// TIA Portal V17 export
// export: Created 2022-12-08T10:14:51.5933257Z, ExportSetting WithDefaults, DisplayName Totally Integrated Automation Portal, DisplayVersion V17 Update 5, DisplayName TIA Portal Openness, DisplayVersion V17 Update 5, DisplayName TIA Portal Version Control Interface, DisplayVersion V17, DisplayName Simotion SCOUT TIA, DisplayVersion 5.4.3.0, DisplayName SINAMICS Startdrive Advanced, DisplayVersion V17 SP1, DisplayName SINAMICS Startdrive G130, G150, S120, S150, SINAMICS MV, S210, DisplayVersion V17 SP1, DisplayName SINAMICS Startdrive G110M, G120, G120C, G120D, G120P, G115D, DisplayVersion V17 SP1, DisplayName STEP 7 Professional, DisplayVersion V17 Update 5, DisplayName STEP 7 Safety, DisplayVersion V17, DisplayName WinCC Advanced, DisplayVersion V17 Update 5
DATA_BLOCK "DB_Glueing"   // DB20
VERSION : 0.1
// stored: AutoNumber true, DBAccessibleFromOPCUA true, DBAccessibleFromWebserver true, InstanceOfName FB_Glueing, InstanceOfType FB
"FB_Glueing"
   // VAR_INPUT
   //    i_Axis : Array["LOWERAXISNUMBER".."UPPERAXISNUMBER"] of DB_ANY;
   //    i_ActualData : Array["LOWERAXISNUMBER".."UPPERAXISNUMBER"] of "UDT_ServoActualData";
   //    i_Reset : Bool;
   //    i_GlueingEnable : Bool;
   //    i_AxesEnabled : Bool;
   //    i_DetectKarton_1 : Bool;
   //    i_DetectKarton_2 : Bool;
   //    i_DetectKarton_3 : Bool;
   //    i_DetectKarton_4 : Bool;
   //    i_DetectKarton_5 : Bool;
   //    i_DetectKarton_6 : Bool;
   //    i_DetectKarton_7 : Bool;
   //    i_DetectKarton_8 : Bool;
   //    i_MasterAxisForGlueing : Int;
   //    i_MaxNumberOfGlueing : Int;
   // END_VAR
   // VAR_OUTPUT
   //    q_TrackOutput_1 : Bool;
   //    q_TrackOutput_2 : Bool;
   //    q_TrackOutput_3 : Bool;
   //    q_TrackOutput_4 : Bool;
   //    q_TrackOutput_5 : Bool;
   //    q_TrackOutput_6 : Bool;
   //    q_TrackOutput_7 : Bool;
   //    q_TrackOutput_8 : Bool;
   //    q_SensorPermanentlyOccupied_1 : Bool;
   //    q_SensorPermanentlyOccupied_2 : Bool;
   //    q_SensorPermanentlyOccupied_3 : Bool;
   //    q_SensorPermanentlyOccupied_4 : Bool;
   //    q_SensorPermanentlyOccupied_5 : Bool;
   //    q_SensorPermanentlyOccupied_6 : Bool;
   //    q_SensorPermanentlyOccupied_7 : Bool;
   //    q_SensorPermanentlyOccupied_8 : Bool;
   //    q_ErrorTechnologyObject : Bool;
   // END_VAR
   // VAR_IN_OUT
   //    iq_Camtracks : Array[1..8] of DB_ANY;
   //    iq_CamData : Array[1..8] of "UDT_Glueing";
   //    iq_OMAC : Array[0.."UPPEROMACMODE"] of "UDT_OMAC_States";
   //    iq_HMIButtons : "UDT_HMI_Buttons";
   // END_VAR
   // VAR
   //    stat_CamValues : Array[1..8] of "FB_Value_CamTrack";
   //    stat_CamCartonDetection { S7_SetPoint := 'True'} : Array[1..8] of "UDT_CamState";
   //    stat_CartonDetectionState { S7_SetPoint := 'True'} : Array[1..8] of Bool;
   //    stat_MCCamTrack { S7_SetPoint := 'True'} : Array[1..8] of MC_CAMTRACK;
   //    stat_ResetCamTrack { S7_SetPoint := 'True'} : Array[1..8] of MC_RESET;
   //    stat_TONSensorPermanentlyOccupied { S7_SetPoint := 'True'} : Array[1..8] of TON_TIME;
   //    stat_SensorPermanentlyOccupied { ExternalAccessible := 'False'; ExternalVisible := 'False'; ExternalWritable := 'False'} : Array[1..8] of Bool;
   //    stat_ErrorTechnologyObject : Bool;
   // END_VAR
BEGIN
END_DATA_BLOCK
